FUNCTION_BLOCK SimOven
VAR
    thermoCouple_Celcius AT %Q* : REAL;
    heaterCurrent_Ampere AT %I* : REAL;
END_VAR
VAR
    previousTemperature : REAL;
    filterParameter : REAL := 0.995;
END_VAR

thermoCouple_Celcius := previousTemperature * filterParameter 
    + LIMIT(20, TO_REAL(EXPT(heaterCurrent_Ampere, 2)), 1E5) * (1 - filterParameter);
previousTemperature := thermoCouple_Celcius;

END_FUNCTION_BLOCK

(* stored: Version 1.1.0.1, ProductVersion 3.1.4024.4
   POU SimOven: Id {bd66a3df-5721-4919-962c-dbbe97ce4652}, SpecialFunc None *)
